// TIA Portal V16 export
// export: Created 2023-03-29T11:03:44.1159531Z, ExportSetting WithDefaults, DisplayName Totally Integrated Automation Portal, DisplayVersion V16 Update 6, DisplayName TIA Portal Version Control Interface, DisplayVersion V16 Update 2, DisplayName TIA Portal Openness, DisplayVersion V16 Update 6, DisplayName STEP 7 Professional, DisplayVersion V16 Update 6, DisplayName STEP 7 Safety, DisplayVersion V16, DisplayName WinCC Advanced, DisplayVersion V16 Update 6
VAR_GLOBAL   // PLC tag table "RTC"
   "memStep_errorMPP04-2" AT %MB103 : USInt;   // bajt pamieci w którym kroku nastąpił błąd modbus
   setErrorModbsmasterMPP04_2 AT %M104.3 : Bool;   // error bit modbus master przepływomierz / Znacznik błedu komunikacji modbus
   "memRisSteperror_MPP04-2" AT %M104.1 : Bool;   // pamięć zbocza dla przechwycenia kroku błedu
   memRisErrorModbusMPP04_2 AT %M104.2 : Bool;   // pamięć zbocza error modbus MPP04-1
   Pobierz_czas AT %M206.2 : Bool;
   Ustaw_czas AT %M206.0 : Bool;
   status_wr_sys_t AT %MW204 : Int;
   status_rd_loc_t AT %MW202 : Int;
   status_rd_sys_t AT %MW200 : Int;
END_VAR
